(* PLC project v0.6.04_CycleSemiAuto.project, CODESYS CODESYS V3.5 SP19 Patch 1 *)
(* stored: creationDateTime 2026-07-22T16:10:21.504862, modificationDateTime 2026-07-22T16:10:21.504862 *)

(* ═══════════════════════════════════════════════════════════════ 🎮 ST_WinchCmd — Commandes IHM pour un Treuil M1/M2 ─────────────────────────────────────────────────────────────── 🎨 Destiné au pilotage manuel et maintenance du treuil depuis l'IHM. ═══════════════════════════════════════════════════════════════ *)
TYPE ST_WinchCmd : STRUCT
  BtnUp : BOOL;  (* ⬆️ Mouvement montee maintenu (mode boutons IHM, MAINT_N1 accessible) *)
  BtnDown : BOOL;  (* ⬇️ Mouvement descente maintenu (mode boutons IHM, MAINT_N1 accessible) *)
  BtnReset : BOOL;  (* 🔑 Demande reset exposée par treuil ; agrégée dans le reset domaine partagé *)
  BtnHome : BOOL;  (* 🎯 Homing nominal si Couplé, unitaire si M1/M2 sélectionné en MAINT_N2 *)
  BtnConfirmCoherence : BOOL;  (* 🔓 Confirmation de cohérence au démarrage *)
  BtnInhibit : BOOL;  (* 🆕 REX 2026-07-08 : bouton IHM inhibition treuil — mise en service, *)
  BtnHomingAtZero : BOOL;  (* 🆕 REX mise en service : force le homing à 0 m (points codeur centre), *)
END_STRUCT;
END_TYPE
